PROGRAM DEADMANCONTROL
VAR
	
	DEADMANCONTROLCASE	:INT; (*CASE STATEMENT*)
	
END_VAR

CASE DEADMANCONTROLCASE	OF
	
(*NORMAL OPERATION*)

	0:
	
	MOBILEHOIST.MAGNETIC_BRAKE1 	:= FALSE;
	MOBILEHOIST.MAGNETIC_BRAKE2 	:= FALSE;
	MOBILEHOIST.SPOTLIGHT			:= FALSE;
	
	IF	MOBILEHOIST.DEADMAN_SWITCH THEN
		
	DEADMANCONTROLCASE :=1;
		
	END_IF
	
(*DEADMAN SWITCH IS PRESSED*)	
	
	1:
	
	IF MOBILEHOIST.DEADMAN_SWITCH THEN
		
		MOBILEHOIST.MAGNETIC_BRAKE1 	:= TRUE;
		MOBILEHOIST.MAGNETIC_BRAKE2 	:= TRUE;
		MOBILEHOIST.SPOTLIGHT			:= TRUE;
		
	ELSE
		
		MOBILEHOIST.MAGNETIC_BRAKE1 	:= FALSE;
		MOBILEHOIST.MAGNETIC_BRAKE2 	:= FALSE;
		MOBILEHOIST.SPOTLIGHT			:= FALSE;
		DEADMANCONTROLCASE 				:= 0;
		
	END_IF

END_CASE

END_PROGRAM

(* stored: Version 1.1.0.1, ProductVersion 3.1.4024.11
   POU DEADMANCONTROL: Id {736eaf38-7d73-476b-a404-94a5aa81a322}, SpecialFunc None *)
